{attribute 'linkalways'} 
{attribute 'no_explicit_call' := 'This FB is a CLASS and must be accessed using methods or properties'}
{attribute 'enable_dynamic_creation'}
FUNCTION_BLOCK FINAL ABS_LWORD EXTENDS Node
VAR
	in : _LWORD(0);
	out : _LWORD(0);
END_VAR

METHOD PUBLIC Clone : I_Node
VAR
	pNode : POINTER TO ABS_LWORD;
END_VAR
pNode := __NEW(ABS_LWORD);
Clone := pNode^;
END_METHOD

METHOD FB_init : BOOL
VAR_INPUT
	bInitRetains : BOOL; // if TRUE, the retain variables are initialized (warm start / cold start)
	bInCopyCode : BOOL;  // if TRUE, the instance afterwards gets moved into the copy code (online change)
END_VAR
AddInput('in',THIS^.in);
AddOutput('out', THIS^.out);
END_METHOD

METHOD PROTECTED OnExecute
VAR
END_VAR
out.Value := ABS(in.Value);
END_METHOD

END_FUNCTION_BLOCK

(* stored: Version 1.1.0.1, ProductVersion 3.1.4024.15
   POU ABS_LWORD: Id {6155d414-552c-40fc-9829-cd90b9d77dd1}, SpecialFunc None
   Folder Constructor: Id {fdf1ad39-74c5-4bcd-b2ce-e82d29b6da06}
   Method Clone: Id {7c6cb390-a34e-45cd-9f6f-1dac4c484aaf}
   Method FB_init: Id {adde9ebb-76f1-4683-90f1-485407f72001}
   Method OnExecute: Id {61438724-5f5a-4859-ab9c-1643e3d9a3d4} *)
